TYPE ST_RxUdpQualisys :
STRUCT
	// Header
	dataSize : UDINT;
	dataType : UDINT;
	timestamp : ULINT;
	frameNumber : UDINT;
	componentCount : UDINT;
	// Component
	componentSize : UDINT;
	componentType : UDINT;
END_STRUCT
END_TYPE

(* stored: Version 1.1.0.1, ProductVersion 3.1.4022.7
   DUT ST_RxUdpQualisys: Id {0593f506-1b48-4a75-b7cf-9cd954548855} *)
